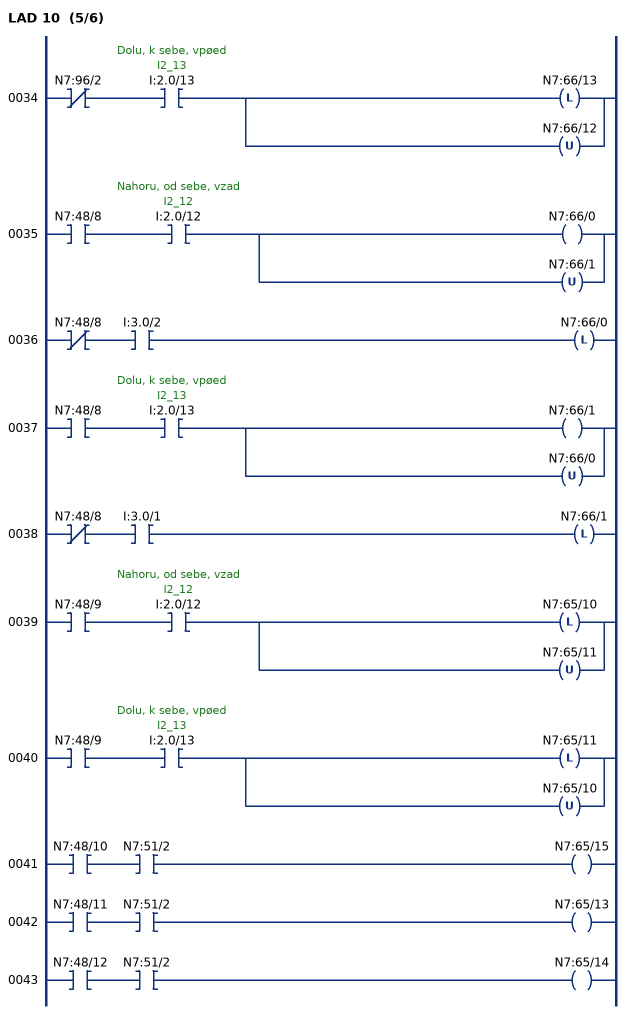
% Rung: 34 %
SOR XIO N7:96/2 XIC I:2.0/13 BST OTL N7:66/13 NXB OTU N7:66/12 BND EOR
%   I:2.0/13  I2_13  "Dolu, k sebe, vpøed" %
% Rung: 35 %
SOR XIC N7:48/8 XIC I:2.0/12 BST OTE N7:66/0 NXB OTU N7:66/1 BND EOR
%   I:2.0/12  I2_12  "Nahoru, od sebe, vzad" %
% Rung: 36 %
SOR XIO N7:48/8 XIC I:3.0/2 OTL N7:66/0 EOR
% Rung: 37 %
SOR XIC N7:48/8 XIC I:2.0/13 BST OTE N7:66/1 NXB OTU N7:66/0 BND EOR
%   I:2.0/13  I2_13  "Dolu, k sebe, vpøed" %
% Rung: 38 %
SOR XIO N7:48/8 XIC I:3.0/1 OTL N7:66/1 EOR
% Rung: 39 %
SOR XIC N7:48/9 XIC I:2.0/12 BST OTL N7:65/10 NXB OTU N7:65/11 BND EOR
%   I:2.0/12  I2_12  "Nahoru, od sebe, vzad" %
% Rung: 40 %
SOR XIC N7:48/9 XIC I:2.0/13 BST OTL N7:65/11 NXB OTU N7:65/10 BND EOR
%   I:2.0/13  I2_13  "Dolu, k sebe, vpøed" %
% Rung: 41 %
SOR XIC N7:48/10 XIC N7:51/2 OTE N7:65/15 EOR
% Rung: 42 %
SOR XIC N7:48/11 XIC N7:51/2 OTE N7:65/13 EOR
% Rung: 43 %
SOR XIC N7:48/12 XIC N7:51/2 OTE N7:65/14 EOR

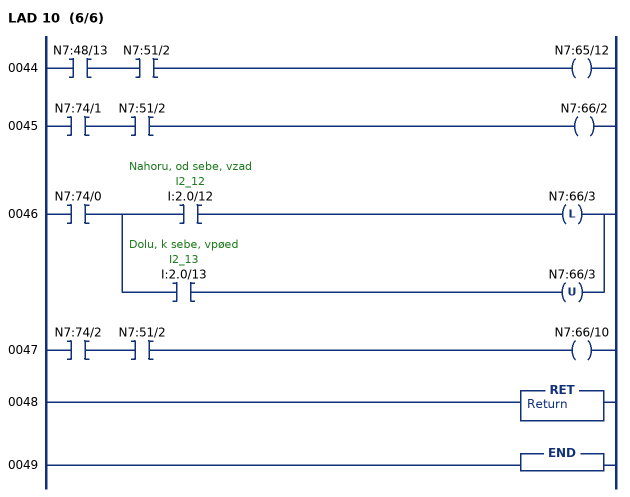
% Rung: 44 %
SOR XIC N7:48/13 XIC N7:51/2 OTE N7:65/12 EOR
% Rung: 45 %
SOR XIC N7:74/1 XIC N7:51/2 OTE N7:66/2 EOR
% Rung: 46 %
SOR XIC N7:74/0 BST XIC I:2.0/12 OTL N7:66/3 NXB XIC I:2.0/13 OTU N7:66/3 BND EOR
%   I:2.0/12  I2_12  "Nahoru, od sebe, vzad" %
%   I:2.0/13  I2_13  "Dolu, k sebe, vpøed" %
% Rung: 47 %
SOR XIC N7:74/2 XIC N7:51/2 OTE N7:66/10 EOR
% Rung: 48 %
SOR RET EOR
% Rung: 49 %
SOR END EOR

LADDER 11
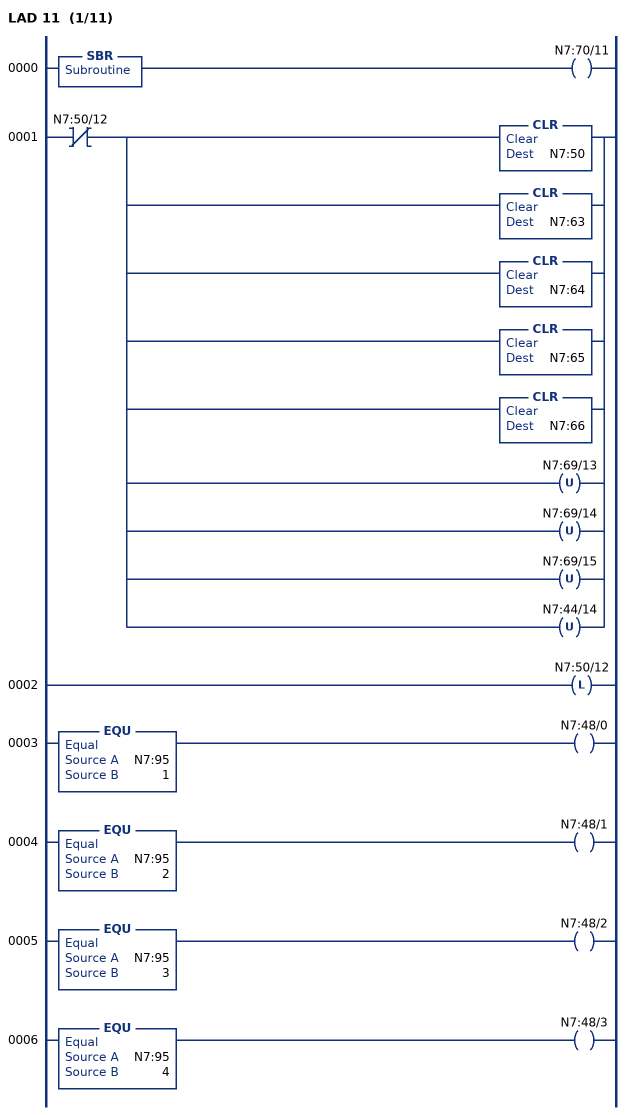
% Rung: 0 %
SOR SBR OTE N7:70/11 EOR
% Rung: 1 %
SOR XIO N7:50/12 BST CLR N7:50 NXB CLR N7:63 NXB CLR N7:64 NXB CLR N7:65 NXB CLR N7:66 NXB OTU N7:69/13 NXB OTU N7:69/14 NXB OTU N7:69/15 NXB OTU N7:44/14 BND EOR
% Rung: 2 %
SOR OTL N7:50/12 EOR
% Rung: 3 %
SOR EQU N7:95 1 OTE N7:48/0 EOR
% Rung: 4 %
SOR EQU N7:95 2 OTE N7:48/1 EOR
% Rung: 5 %
SOR EQU N7:95 3 OTE N7:48/2 EOR
% Rung: 6 %
SOR EQU N7:95 4 OTE N7:48/3 EOR

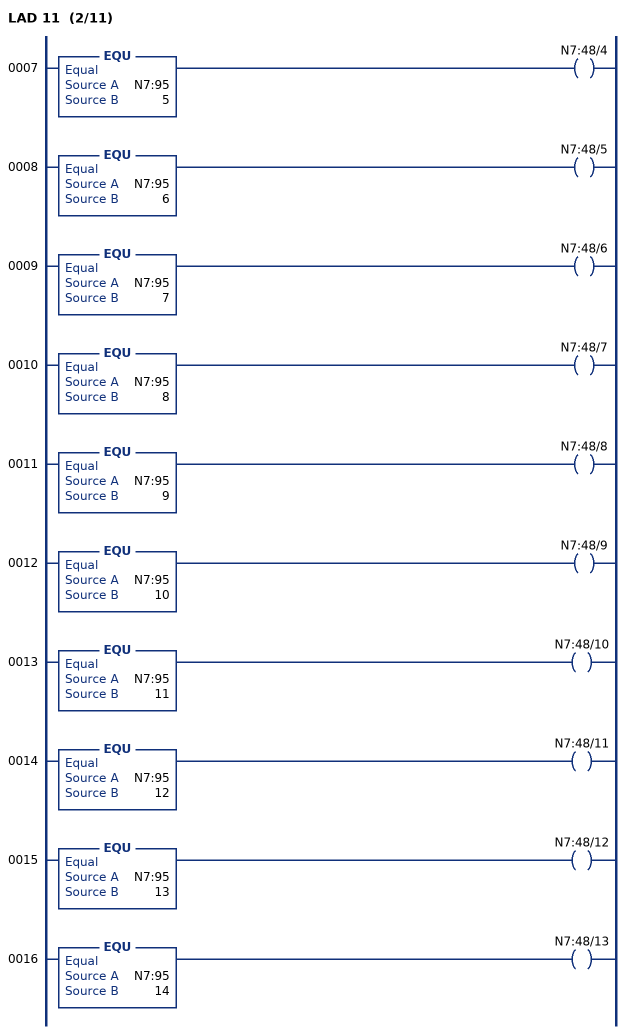
% Rung: 7 %
SOR EQU N7:95 5 OTE N7:48/4 EOR
% Rung: 8 %
SOR EQU N7:95 6 OTE N7:48/5 EOR
% Rung: 9 %
SOR EQU N7:95 7 OTE N7:48/6 EOR
% Rung: 10 %
SOR EQU N7:95 8 OTE N7:48/7 EOR
% Rung: 11 %
SOR EQU N7:95 9 OTE N7:48/8 EOR
% Rung: 12 %
SOR EQU N7:95 10 OTE N7:48/9 EOR
% Rung: 13 %
SOR EQU N7:95 11 OTE N7:48/10 EOR
% Rung: 14 %
SOR EQU N7:95 12 OTE N7:48/11 EOR
% Rung: 15 %
SOR EQU N7:95 13 OTE N7:48/12 EOR
% Rung: 16 %
SOR EQU N7:95 14 OTE N7:48/13 EOR

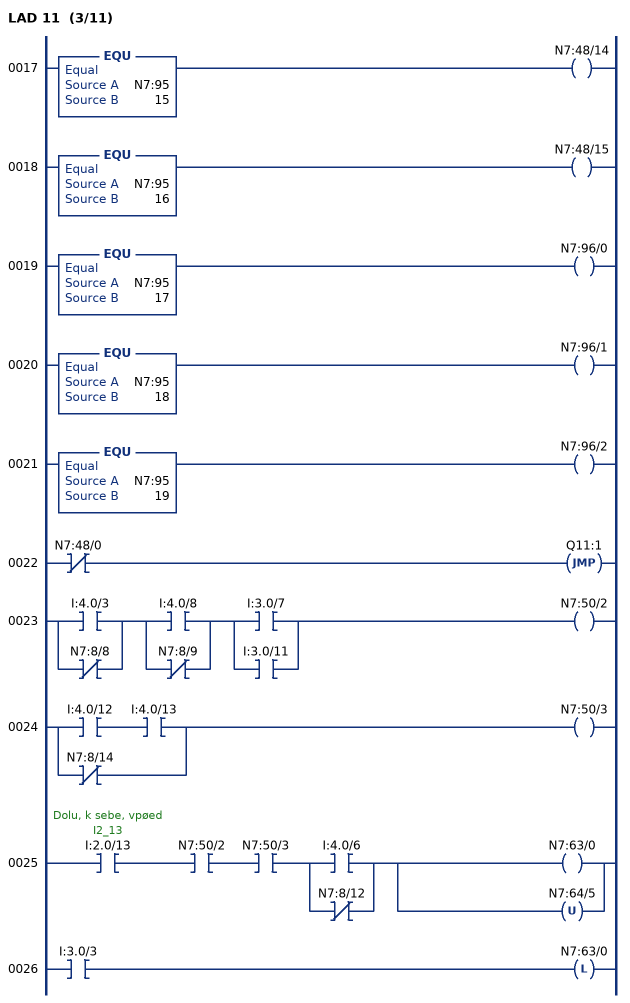
% Rung: 17 %
SOR EQU N7:95 15 OTE N7:48/14 EOR
% Rung: 18 %
SOR EQU N7:95 16 OTE N7:48/15 EOR
% Rung: 19 %
SOR EQU N7:95 17 OTE N7:96/0 EOR
% Rung: 20 %
SOR EQU N7:95 18 OTE N7:96/1 EOR
% Rung: 21 %
SOR EQU N7:95 19 OTE N7:96/2 EOR
% Rung: 22 %
SOR XIO N7:48/0 JMP Q11:1 EOR
% Rung: 23 %
SOR BST XIC I:4.0/3 NXB XIO N7:8/8 BND BST XIC I:4.0/8 NXB XIO N7:8/9 BND BST XIC I:3.0/7 NXB XIC I:3.0/11 BND OTE N7:50/2 EOR
% Rung: 24 %
SOR BST XIC I:4.0/12 XIC I:4.0/13 NXB XIO N7:8/14 BND OTE N7:50/3 EOR
% Rung: 25 %
SOR XIC I:2.0/13 XIC N7:50/2 XIC N7:50/3 BST XIC I:4.0/6 NXB XIO N7:8/12 BND BST OTE N7:63/0 NXB OTU N7:64/5 BND EOR
%   I:2.0/13  I2_13  "Dolu, k sebe, vpøed" %
% Rung: 26 %
SOR XIC I:3.0/3 OTL N7:63/0 EOR

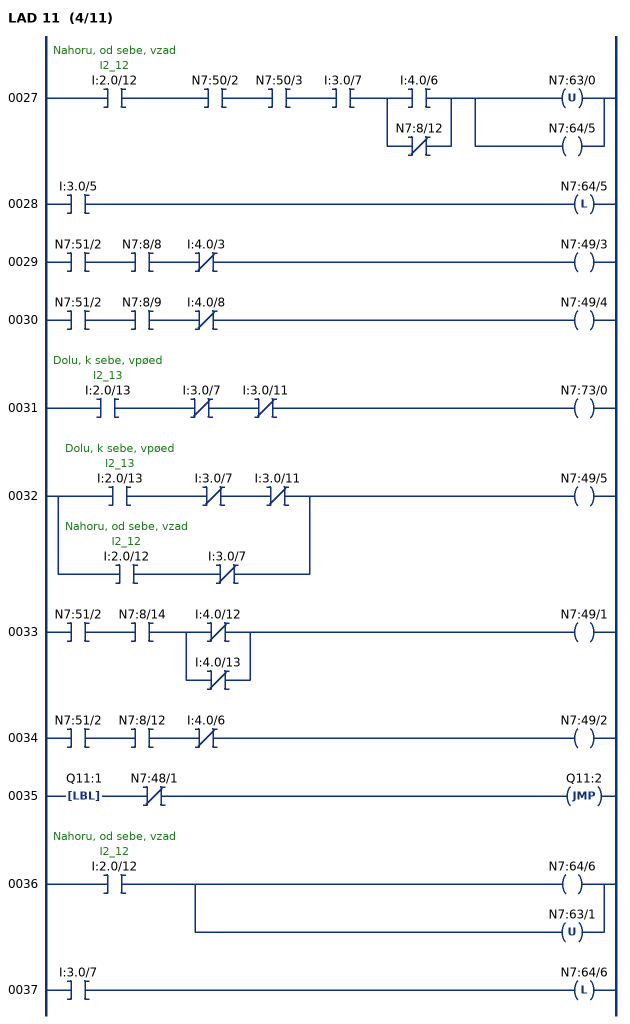
% Rung: 27 %
SOR XIC I:2.0/12 XIC N7:50/2 XIC N7:50/3 XIC I:3.0/7 BST XIC I:4.0/6 NXB XIO N7:8/12 BND BST OTU N7:63/0 NXB OTE N7:64/5 BND EOR
%   I:2.0/12  I2_12  "Nahoru, od sebe, vzad" %
% Rung: 28 %
SOR XIC I:3.0/5 OTL N7:64/5 EOR
% Rung: 29 %
SOR XIC N7:51/2 XIC N7:8/8 XIO I:4.0/3 OTE N7:49/3 EOR
% Rung: 30 %
SOR XIC N7:51/2 XIC N7:8/9 XIO I:4.0/8 OTE N7:49/4 EOR
% Rung: 31 %
SOR XIC I:2.0/13 XIO I:3.0/7 XIO I:3.0/11 OTE N7:73/0 EOR
%   I:2.0/13  I2_13  "Dolu, k sebe, vpøed" %
% Rung: 32 %
SOR BST XIC I:2.0/13 XIO I:3.0/7 XIO I:3.0/11 NXB XIC I:2.0/12 XIO I:3.0/7 BND OTE N7:49/5 EOR
%   I:2.0/13  I2_13  "Dolu, k sebe, vpøed" %
%   I:2.0/12  I2_12  "Nahoru, od sebe, vzad" %
% Rung: 33 %
SOR XIC N7:51/2 XIC N7:8/14 BST XIO I:4.0/12 NXB XIO I:4.0/13 BND OTE N7:49/1 EOR
% Rung: 34 %
SOR XIC N7:51/2 XIC N7:8/12 XIO I:4.0/6 OTE N7:49/2 EOR
% Rung: 35 %
SOR LBL Q11:1 XIO N7:48/1 JMP Q11:2 EOR
% Rung: 36 %
SOR XIC I:2.0/12 BST OTE N7:64/6 NXB OTU N7:63/1 BND EOR
%   I:2.0/12  I2_12  "Nahoru, od sebe, vzad" %
% Rung: 37 %
SOR XIC I:3.0/7 OTL N7:64/6 EOR

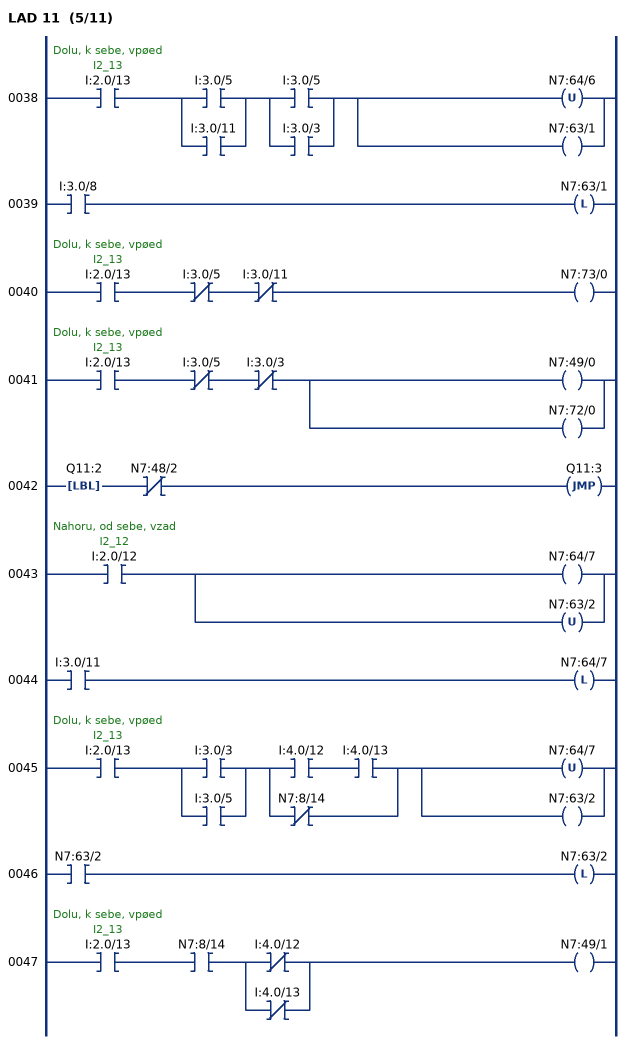
% Rung: 38 %
SOR XIC I:2.0/13 BST XIC I:3.0/5 NXB XIC I:3.0/11 BND BST XIC I:3.0/5 NXB XIC I:3.0/3 BND BST OTU N7:64/6 NXB OTE N7:63/1 BND EOR
%   I:2.0/13  I2_13  "Dolu, k sebe, vpøed" %
% Rung: 39 %
SOR XIC I:3.0/8 OTL N7:63/1 EOR
% Rung: 40 %
SOR XIC I:2.0/13 XIO I:3.0/5 XIO I:3.0/11 OTE N7:73/0 EOR
%   I:2.0/13  I2_13  "Dolu, k sebe, vpøed" %
% Rung: 41 %
SOR XIC I:2.0/13 XIO I:3.0/5 XIO I:3.0/3 BST OTE N7:49/0 NXB OTE N7:72/0 BND EOR
%   I:2.0/13  I2_13  "Dolu, k sebe, vpøed" %
% Rung: 42 %
SOR LBL Q11:2 XIO N7:48/2 JMP Q11:3 EOR
% Rung: 43 %
SOR XIC I:2.0/12 BST OTE N7:64/7 NXB OTU N7:63/2 BND EOR
%   I:2.0/12  I2_12  "Nahoru, od sebe, vzad" %
% Rung: 44 %
SOR XIC I:3.0/11 OTL N7:64/7 EOR
% Rung: 45 %
SOR XIC I:2.0/13 BST XIC I:3.0/3 NXB XIC I:3.0/5 BND BST XIC I:4.0/12 XIC I:4.0/13 NXB XIO N7:8/14 BND BST OTU N7:64/7 NXB OTE N7:63/2 BND EOR
%   I:2.0/13  I2_13  "Dolu, k sebe, vpøed" %
% Rung: 46 %
SOR XIC N7:63/2 OTL N7:63/2 EOR
% Rung: 47 %
SOR XIC I:2.0/13 XIC N7:8/14 BST XIO I:4.0/12 NXB XIO I:4.0/13 BND OTE N7:49/1 EOR
%   I:2.0/13  I2_13  "Dolu, k sebe, vpøed" %

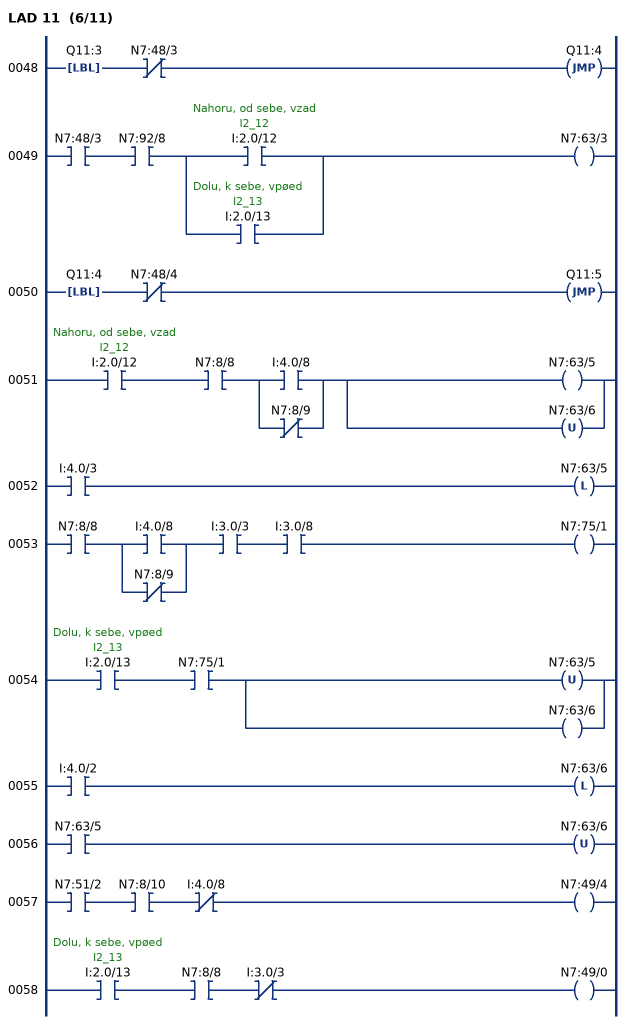
% Rung: 48 %
SOR LBL Q11:3 XIO N7:48/3 JMP Q11:4 EOR
% Rung: 49 %
SOR XIC N7:48/3 XIC N7:92/8 BST XIC I:2.0/12 NXB XIC I:2.0/13 BND OTE N7:63/3 EOR
%   I:2.0/12  I2_12  "Nahoru, od sebe, vzad" %
%   I:2.0/13  I2_13  "Dolu, k sebe, vpøed" %
% Rung: 50 %
SOR LBL Q11:4 XIO N7:48/4 JMP Q11:5 EOR
% Rung: 51 %
SOR XIC I:2.0/12 XIC N7:8/8 BST XIC I:4.0/8 NXB XIO N7:8/9 BND BST OTE N7:63/5 NXB OTU N7:63/6 BND EOR
%   I:2.0/12  I2_12  "Nahoru, od sebe, vzad" %
% Rung: 52 %
SOR XIC I:4.0/3 OTL N7:63/5 EOR
% Rung: 53 %
SOR XIC N7:8/8 BST XIC I:4.0/8 NXB XIO N7:8/9 BND XIC I:3.0/3 XIC I:3.0/8 OTE N7:75/1 EOR
% Rung: 54 %
SOR XIC I:2.0/13 XIC N7:75/1 BST OTU N7:63/5 NXB OTE N7:63/6 BND EOR
%   I:2.0/13  I2_13  "Dolu, k sebe, vpøed" %
% Rung: 55 %
SOR XIC I:4.0/2 OTL N7:63/6 EOR
% Rung: 56 %
SOR XIC N7:63/5 OTU N7:63/6 EOR
% Rung: 57 %
SOR XIC N7:51/2 XIC N7:8/10 XIO I:4.0/8 OTE N7:49/4 EOR
% Rung: 58 %
SOR XIC I:2.0/13 XIC N7:8/8 XIO I:3.0/3 OTE N7:49/0 EOR
%   I:2.0/13  I2_13  "Dolu, k sebe, vpøed" %

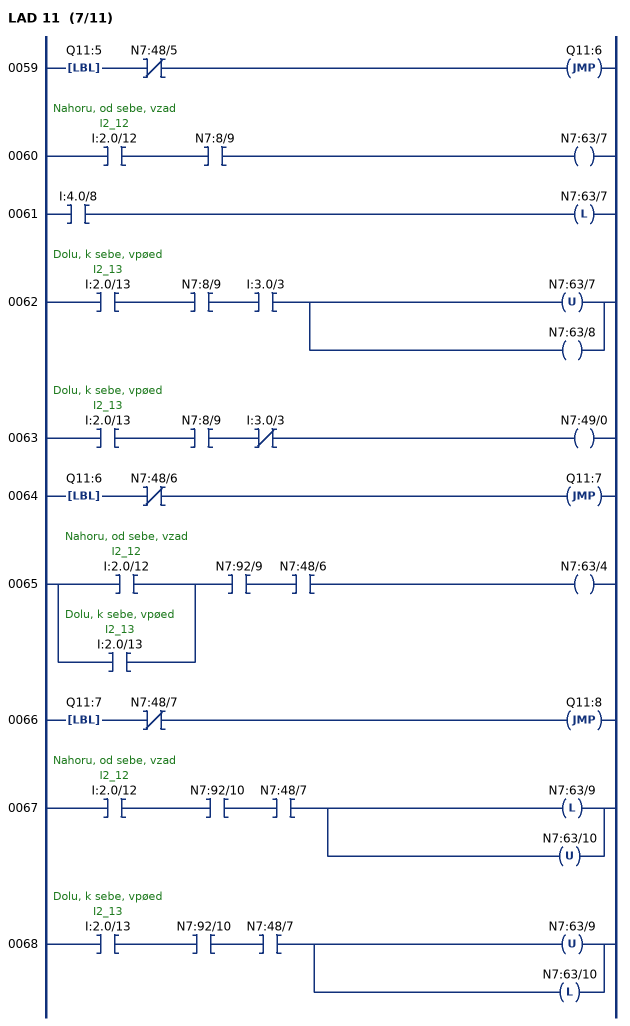
% Rung: 59 %
SOR LBL Q11:5 XIO N7:48/5 JMP Q11:6 EOR
% Rung: 60 %
SOR XIC I:2.0/12 XIC N7:8/9 OTE N7:63/7 EOR
%   I:2.0/12  I2_12  "Nahoru, od sebe, vzad" %
% Rung: 61 %
SOR XIC I:4.0/8 OTL N7:63/7 EOR
% Rung: 62 %
SOR XIC I:2.0/13 XIC N7:8/9 XIC I:3.0/3 BST OTU N7:63/7 NXB OTE N7:63/8 BND EOR
%   I:2.0/13  I2_13  "Dolu, k sebe, vpøed" %
% Rung: 63 %
SOR XIC I:2.0/13 XIC N7:8/9 XIO I:3.0/3 OTE N7:49/0 EOR
%   I:2.0/13  I2_13  "Dolu, k sebe, vpøed" %
% Rung: 64 %
SOR LBL Q11:6 XIO N7:48/6 JMP Q11:7 EOR
% Rung: 65 %
SOR BST XIC I:2.0/12 NXB XIC I:2.0/13 BND XIC N7:92/9 XIC N7:48/6 OTE N7:63/4 EOR
%   I:2.0/12  I2_12  "Nahoru, od sebe, vzad" %
%   I:2.0/13  I2_13  "Dolu, k sebe, vpøed" %
% Rung: 66 %
SOR LBL Q11:7 XIO N7:48/7 JMP Q11:8 EOR
% Rung: 67 %
SOR XIC I:2.0/12 XIC N7:92/10 XIC N7:48/7 BST OTL N7:63/9 NXB OTU N7:63/10 BND EOR
%   I:2.0/12  I2_12  "Nahoru, od sebe, vzad" %
% Rung: 68 %
SOR XIC I:2.0/13 XIC N7:92/10 XIC N7:48/7 BST OTU N7:63/9 NXB OTL N7:63/10 BND EOR
%   I:2.0/13  I2_13  "Dolu, k sebe, vpøed" %

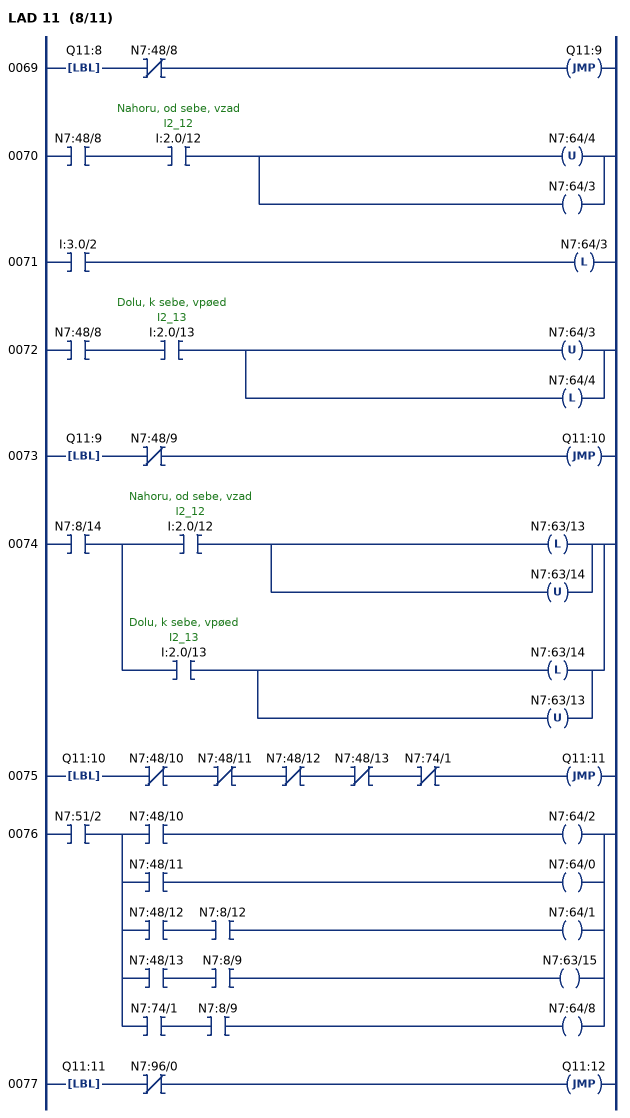
% Rung: 69 %
SOR LBL Q11:8 XIO N7:48/8 JMP Q11:9 EOR
% Rung: 70 %
SOR XIC N7:48/8 XIC I:2.0/12 BST OTU N7:64/4 NXB OTE N7:64/3 BND EOR
%   I:2.0/12  I2_12  "Nahoru, od sebe, vzad" %
% Rung: 71 %
SOR XIC I:3.0/2 OTL N7:64/3 EOR
% Rung: 72 %
SOR XIC N7:48/8 XIC I:2.0/13 BST OTU N7:64/3 NXB OTL N7:64/4 BND EOR
%   I:2.0/13  I2_13  "Dolu, k sebe, vpøed" %
% Rung: 73 %
SOR LBL Q11:9 XIO N7:48/9 JMP Q11:10 EOR
% Rung: 74 %
SOR XIC N7:8/14 BST XIC I:2.0/12 BST OTL N7:63/13 NXB OTU N7:63/14 BND NXB XIC I:2.0/13 BST OTL N7:63/14 NXB OTU N7:63/13 BND BND EOR
%   I:2.0/12  I2_12  "Nahoru, od sebe, vzad" %
%   I:2.0/13  I2_13  "Dolu, k sebe, vpøed" %
% Rung: 75 %
SOR LBL Q11:10 XIO N7:48/10 XIO N7:48/11 XIO N7:48/12 XIO N7:48/13 XIO N7:74/1 JMP Q11:11 EOR
% Rung: 76 %
SOR XIC N7:51/2 BST XIC N7:48/10 OTE N7:64/2 NXB BST XIC N7:48/11 OTE N7:64/0 NXB XIC N7:48/12 XIC N7:8/12 OTE N7:64/1 NXB XIC N7:48/13 XIC N7:8/9 OTE N7:63/15 NXB XIC N7:74/1 XIC N7:8/9 OTE N7:64/8 BND BND EOR
% Rung: 77 %
SOR LBL Q11:11 XIO N7:96/0 JMP Q11:12 EOR

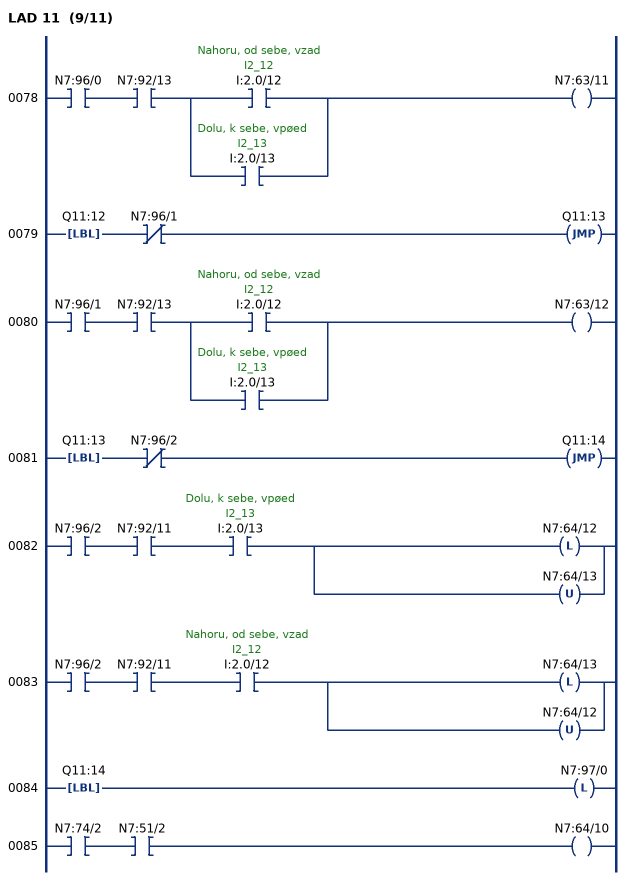
% Rung: 78 %
SOR XIC N7:96/0 XIC N7:92/13 BST XIC I:2.0/12 NXB XIC I:2.0/13 BND OTE N7:63/11 EOR
%   I:2.0/12  I2_12  "Nahoru, od sebe, vzad" %
%   I:2.0/13  I2_13  "Dolu, k sebe, vpøed" %
% Rung: 79 %
SOR LBL Q11:12 XIO N7:96/1 JMP Q11:13 EOR
% Rung: 80 %
SOR XIC N7:96/1 XIC N7:92/13 BST XIC I:2.0/12 NXB XIC I:2.0/13 BND OTE N7:63/12 EOR
%   I:2.0/12  I2_12  "Nahoru, od sebe, vzad" %
%   I:2.0/13  I2_13  "Dolu, k sebe, vpøed" %
% Rung: 81 %
SOR LBL Q11:13 XIO N7:96/2 JMP Q11:14 EOR
% Rung: 82 %
SOR XIC N7:96/2 XIC N7:92/11 XIC I:2.0/13 BST OTL N7:64/12 NXB OTU N7:64/13 BND EOR
%   I:2.0/13  I2_13  "Dolu, k sebe, vpøed" %
% Rung: 83 %
SOR XIC N7:96/2 XIC N7:92/11 XIC I:2.0/12 BST OTL N7:64/13 NXB OTU N7:64/12 BND EOR
%   I:2.0/12  I2_12  "Nahoru, od sebe, vzad" %
% Rung: 84 %
SOR LBL Q11:14 OTL N7:97/0 EOR
% Rung: 85 %
SOR XIC N7:74/2 XIC N7:51/2 OTE N7:64/10 EOR

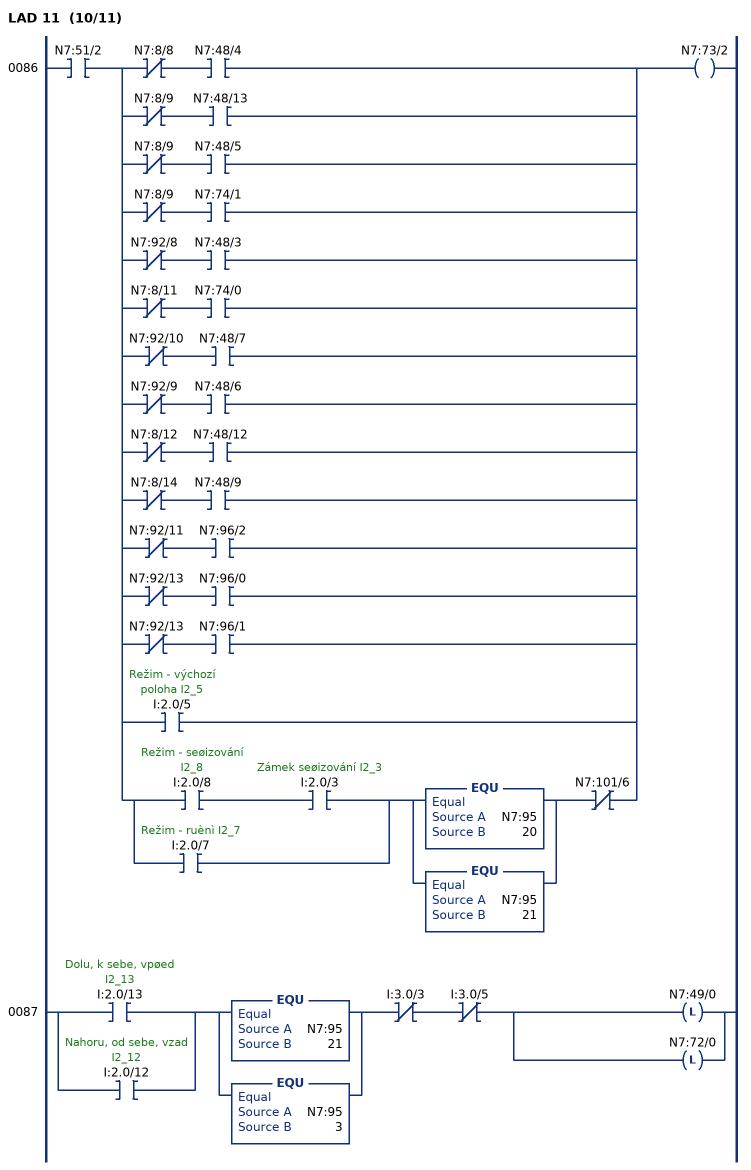
% Rung: 86 %
SOR XIC N7:51/2 BST XIO N7:8/8 XIC N7:48/4 NXB XIO N7:8/9 XIC N7:48/13 NXB XIO N7:8/9 XIC N7:48/5 NXB XIO N7:8/9 XIC N7:74/1 NXB XIO N7:92/8 XIC N7:48/3 NXB XIO N7:8/11 XIC N7:74/0 NXB XIO N7:92/10 XIC N7:48/7 NXB XIO N7:92/9 XIC N7:48/6 NXB XIO N7:8/12 XIC N7:48/12 NXB BST BST BST XIO N7:8/14 XIC N7:48/9 NXB XIO N7:92/11 XIC N7:96/2 BND NXB XIO N7:92/13 XIC N7:96/0 BND NXB XIO N7:92/13 XIC N7:96/1 NXB BST XIC I:2.0/5 NXB BST XIC I:2.0/8 XIC I:2.0/3 NXB XIC I:2.0/7 BND BST EQU N7:95 20 NXB EQU N7:95 21 BND XIO N7:101/6 BND BND BND OTE N7:73/2 EOR
%   I:2.0/5  I2_5  "Režim - výchozí poloha" %
%   I:2.0/8  I2_8  "Režim - seøizování" %
%   I:2.0/3  I2_3  "Zámek seøizování" %
%   I:2.0/7  I2_7  "Režim - ruènì" %
% Rung: 87 %
SOR BST XIC I:2.0/13 NXB XIC I:2.0/12 BND BST EQU N7:95 21 NXB EQU N7:95 3 BND XIO I:3.0/3 XIO I:3.0/5 BST OTL N7:49/0 NXB OTL N7:72/0 BND EOR
%   I:2.0/13  I2_13  "Dolu, k sebe, vpøed" %
%   I:2.0/12  I2_12  "Nahoru, od sebe, vzad" %

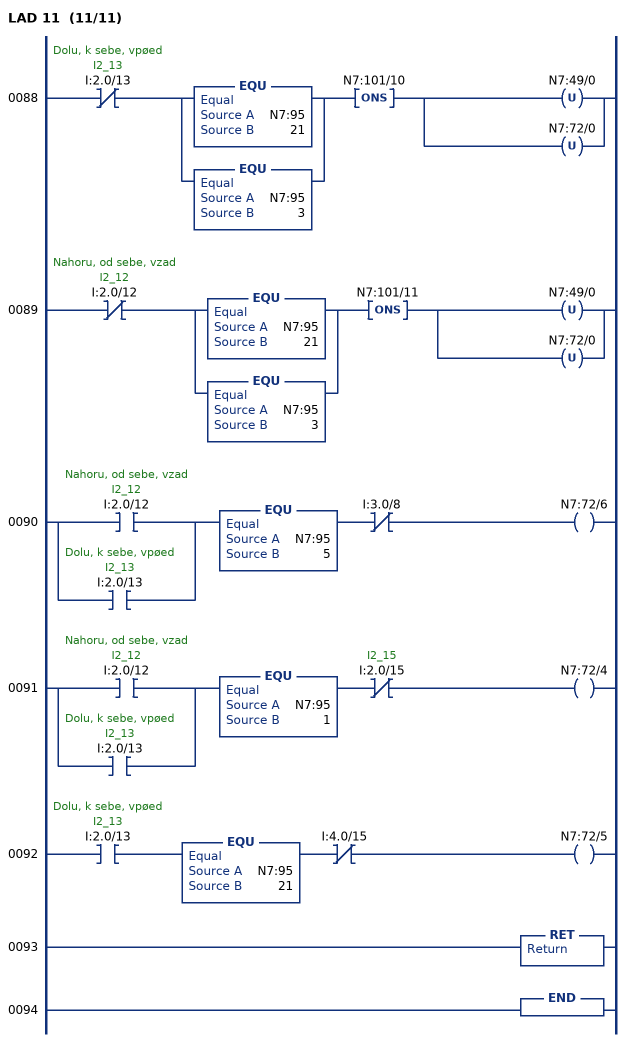
% Rung: 88 %
SOR XIO I:2.0/13 BST EQU N7:95 21 NXB EQU N7:95 3 BND OSR N7:101/10 BST OTU N7:49/0 NXB OTU N7:72/0 BND EOR
%   I:2.0/13  I2_13  "Dolu, k sebe, vpøed" %
% Rung: 89 %
SOR XIO I:2.0/12 BST EQU N7:95 21 NXB EQU N7:95 3 BND OSR N7:101/11 BST OTU N7:49/0 NXB OTU N7:72/0 BND EOR
%   I:2.0/12  I2_12  "Nahoru, od sebe, vzad" %
% Rung: 90 %
SOR BST XIC I:2.0/12 NXB XIC I:2.0/13 BND EQU N7:95 5 XIO I:3.0/8 OTE N7:72/6 EOR
%   I:2.0/12  I2_12  "Nahoru, od sebe, vzad" %
%   I:2.0/13  I2_13  "Dolu, k sebe, vpøed" %
% Rung: 91 %
SOR BST XIC I:2.0/12 NXB XIC I:2.0/13 BND EQU N7:95 1 XIO I:2.0/15 OTE N7:72/4 EOR
%   I:2.0/12  I2_12  "Nahoru, od sebe, vzad" %
%   I:2.0/13  I2_13  "Dolu, k sebe, vpøed" %
%   I:2.0/15  I2_15 %
% Rung: 92 %
SOR XIC I:2.0/13 EQU N7:95 21 XIO I:4.0/15 OTE N7:72/5 EOR
%   I:2.0/13  I2_13  "Dolu, k sebe, vpøed" %
% Rung: 93 %
SOR RET EOR
% Rung: 94 %
SOR END EOR

LADDER 12
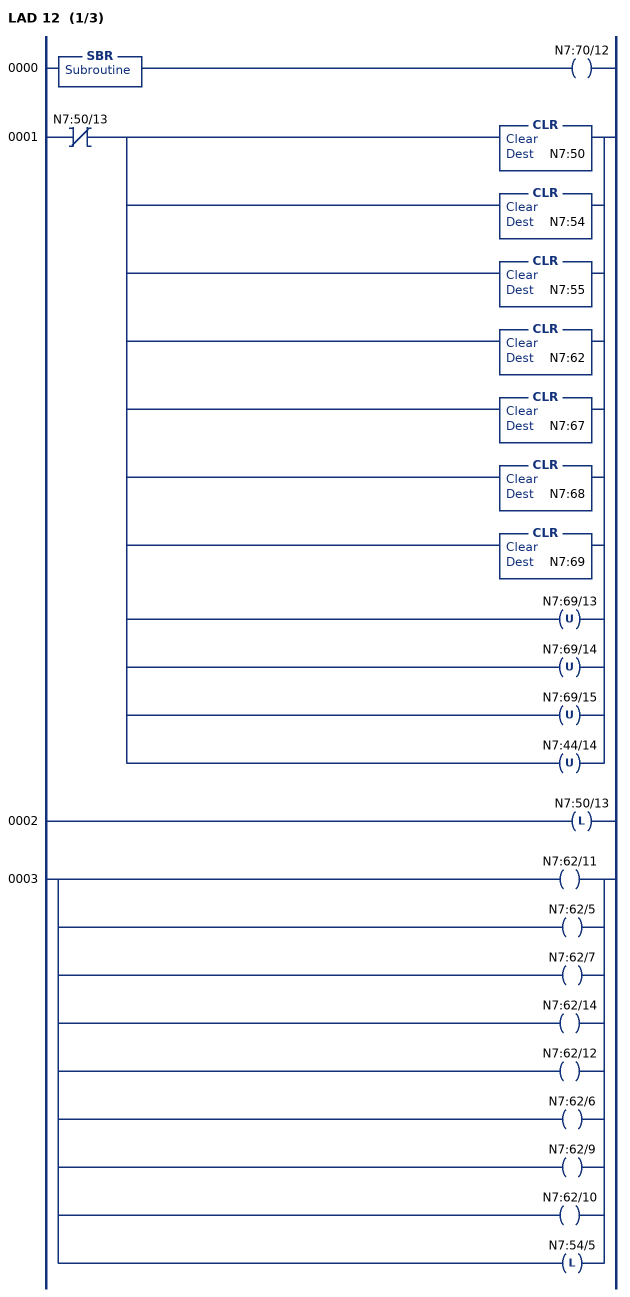
% Rung: 0 %
SOR SBR OTE N7:70/12 EOR
% Rung: 1 %
SOR XIO N7:50/13 BST CLR N7:50 NXB CLR N7:54 NXB CLR N7:55 NXB CLR N7:62 NXB CLR N7:67 NXB CLR N7:68 NXB CLR N7:69 NXB OTU N7:69/13 NXB OTU N7:69/14 NXB OTU N7:69/15 NXB OTU N7:44/14 BND EOR
% Rung: 2 %
SOR OTL N7:50/13 EOR
% Rung: 3 %
SOR BST OTE N7:62/11 NXB OTE N7:62/5 NXB OTE N7:62/7 NXB OTE N7:62/14 NXB BST OTE N7:62/12 NXB OTE N7:62/6 BND NXB OTE N7:62/9 NXB OTE N7:62/10 NXB OTL N7:54/5 BND EOR

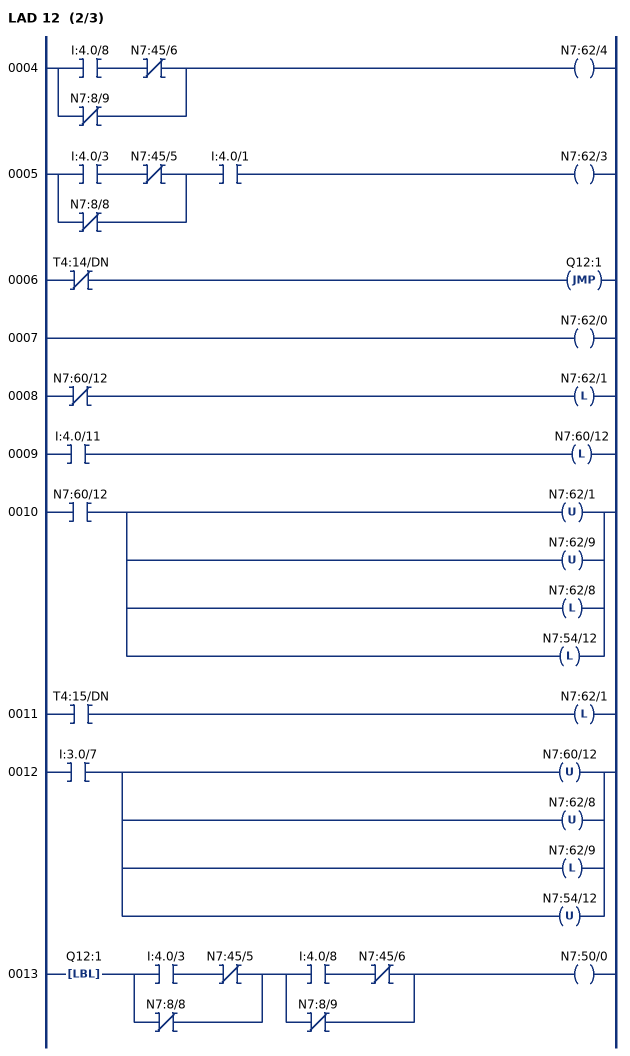
% Rung: 4 %
SOR BST XIC I:4.0/8 XIO N7:45/6 NXB XIO N7:8/9 BND OTE N7:62/4 EOR
% Rung: 5 %
SOR BST XIC I:4.0/3 XIO N7:45/5 NXB XIO N7:8/8 BND XIC I:4.0/1 OTE N7:62/3 EOR
% Rung: 6 %
SOR XIO T4:14/DN JMP Q12:1 EOR
% Rung: 7 %
SOR OTE N7:62/0 EOR
% Rung: 8 %
SOR XIO N7:60/12 OTL N7:62/1 EOR
% Rung: 9 %
SOR XIC I:4.0/11 OTL N7:60/12 EOR
% Rung: 10 %
SOR XIC N7:60/12 BST OTU N7:62/1 NXB BST OTU N7:62/9 NXB OTL N7:62/8 NXB OTL N7:54/12 BND BND EOR
% Rung: 11 %
SOR XIC T4:15/DN OTL N7:62/1 EOR
% Rung: 12 %
SOR XIC I:3.0/7 BST OTU N7:60/12 NXB OTU N7:62/8 NXB OTL N7:62/9 NXB OTU N7:54/12 BND EOR
% Rung: 13 %
SOR LBL Q12:1 BST XIC I:4.0/3 XIO N7:45/5 NXB XIO N7:8/8 BND BST XIC I:4.0/8 XIO N7:45/6 NXB XIO N7:8/9 BND OTE N7:50/0 EOR

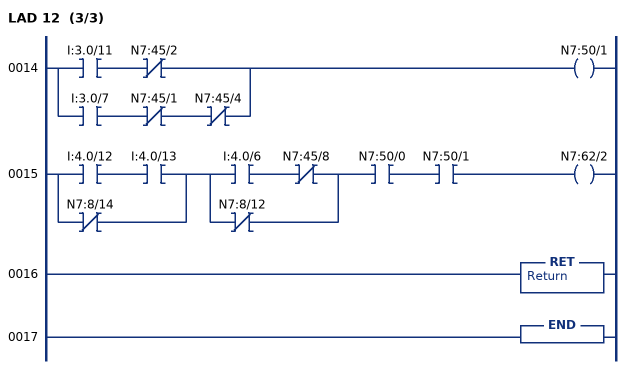
% Rung: 14 %
SOR BST XIC I:3.0/11 XIO N7:45/2 NXB XIC I:3.0/7 XIO N7:45/1 XIO N7:45/4 BND OTE N7:50/1 EOR
% Rung: 15 %
SOR BST XIC I:4.0/12 XIC I:4.0/13 NXB XIO N7:8/14 BND BST XIC I:4.0/6 XIO N7:45/8 NXB XIO N7:8/12 BND XIC N7:50/0 XIC N7:50/1 OTE N7:62/2 EOR
% Rung: 16 %
SOR RET EOR
% Rung: 17 %
SOR END EOR

LADDER 13
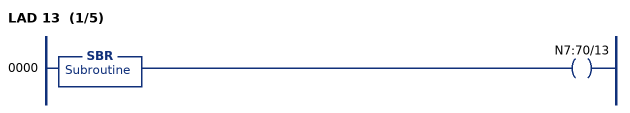
% Rung: 0 %
SOR SBR OTE N7:70/13 EOR

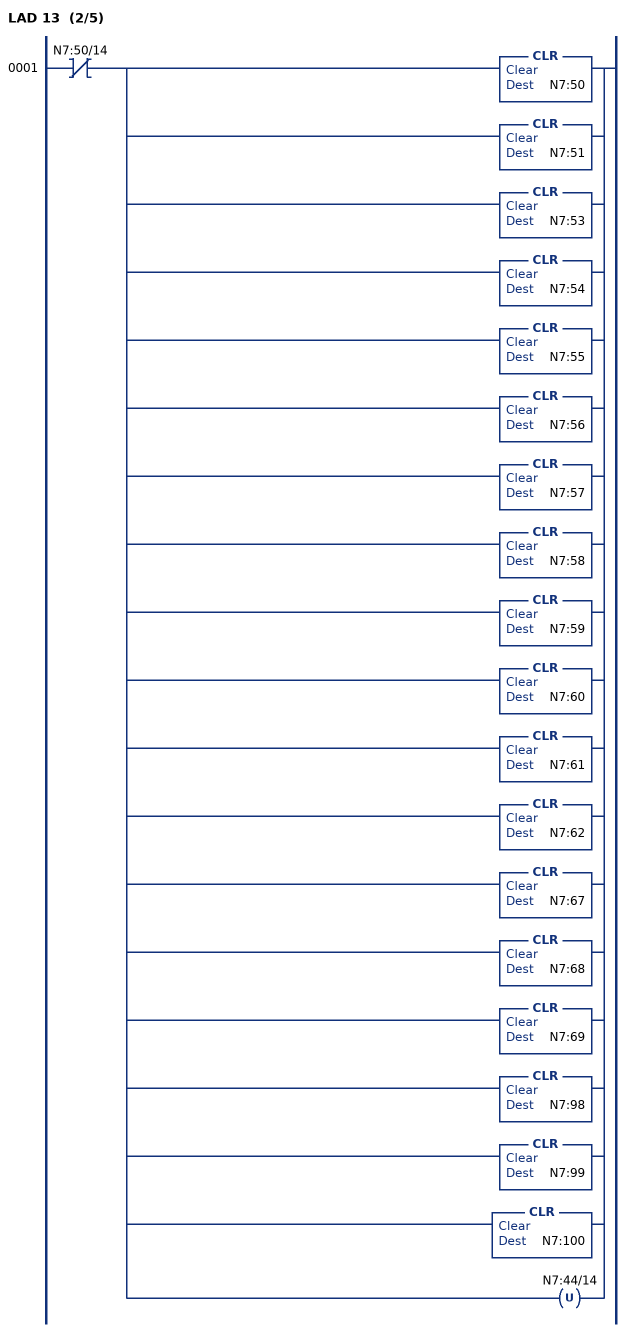
% Rung: 1 %
SOR XIO N7:50/14 BST CLR N7:50 NXB CLR N7:51 NXB CLR N7:53 NXB CLR N7:54 NXB CLR N7:55 NXB CLR N7:56 NXB CLR N7:57 NXB CLR N7:58 NXB CLR N7:59 NXB CLR N7:60 NXB CLR N7:61 NXB CLR N7:62 NXB CLR N7:67 NXB CLR N7:68 NXB BST BST CLR N7:69 NXB CLR N7:98 BND NXB BST CLR N7:99 NXB CLR N7:100 BND BND NXB OTU N7:44/14 BND EOR

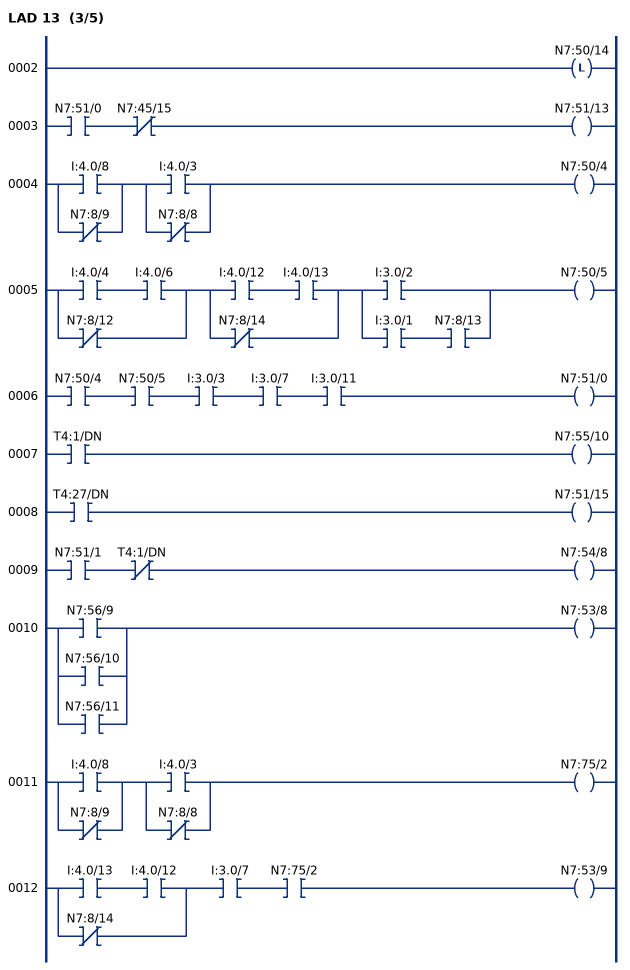
% Rung: 2 %
SOR OTL N7:50/14 EOR
% Rung: 3 %
SOR XIC N7:51/0 XIO N7:45/15 OTE N7:51/13 EOR
% Rung: 4 %
SOR BST XIC I:4.0/8 NXB XIO N7:8/9 BND BST XIC I:4.0/3 NXB XIO N7:8/8 BND OTE N7:50/4 EOR
% Rung: 5 %
SOR BST XIC I:4.0/4 XIC I:4.0/6 NXB XIO N7:8/12 BND BST XIC I:4.0/12 XIC I:4.0/13 NXB XIO N7:8/14 BND BST XIC I:3.0/2 NXB XIC I:3.0/1 XIC N7:8/13 BND OTE N7:50/5 EOR
% Rung: 6 %
SOR XIC N7:50/4 XIC N7:50/5 XIC I:3.0/3 XIC I:3.0/7 XIC I:3.0/11 OTE N7:51/0 EOR
% Rung: 7 %
SOR XIC T4:1/DN OTE N7:55/10 EOR
% Rung: 8 %
SOR XIC T4:27/DN OTE N7:51/15 EOR
% Rung: 9 %
SOR XIC N7:51/1 XIO T4:1/DN OTE N7:54/8 EOR
% Rung: 10 %
SOR BST XIC N7:56/9 NXB XIC N7:56/10 NXB XIC N7:56/11 BND OTE N7:53/8 EOR
% Rung: 11 %
SOR BST XIC I:4.0/8 NXB XIO N7:8/9 BND BST XIC I:4.0/3 NXB XIO N7:8/8 BND OTE N7:75/2 EOR
% Rung: 12 %
SOR BST XIC I:4.0/13 XIC I:4.0/12 NXB XIO N7:8/14 BND XIC I:3.0/7 XIC N7:75/2 OTE N7:53/9 EOR

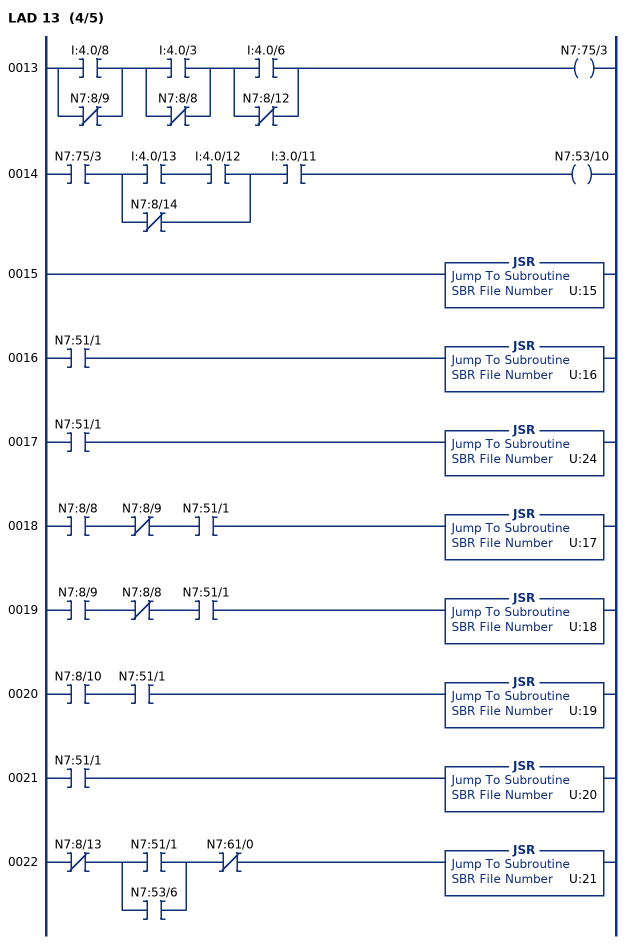
% Rung: 13 %
SOR BST XIC I:4.0/8 NXB XIO N7:8/9 BND BST XIC I:4.0/3 NXB XIO N7:8/8 BND BST XIC I:4.0/6 NXB XIO N7:8/12 BND OTE N7:75/3 EOR
% Rung: 14 %
SOR XIC N7:75/3 BST XIC I:4.0/13 XIC I:4.0/12 NXB XIO N7:8/14 BND XIC I:3.0/11 OTE N7:53/10 EOR
% Rung: 15 %
SOR JSR U:15 EOR
% Rung: 16 %
SOR XIC N7:51/1 JSR U:16 EOR
% Rung: 17 %
SOR XIC N7:51/1 JSR U:24 EOR
% Rung: 18 %
SOR XIC N7:8/8 XIO N7:8/9 XIC N7:51/1 JSR U:17 EOR
% Rung: 19 %
SOR XIC N7:8/9 XIO N7:8/8 XIC N7:51/1 JSR U:18 EOR
% Rung: 20 %
SOR XIC N7:8/10 XIC N7:51/1 JSR U:19 EOR
% Rung: 21 %
SOR XIC N7:51/1 JSR U:20 EOR
% Rung: 22 %
SOR XIO N7:8/13 BST XIC N7:51/1 NXB XIC N7:53/6 BND XIO N7:61/0 JSR U:21 EOR

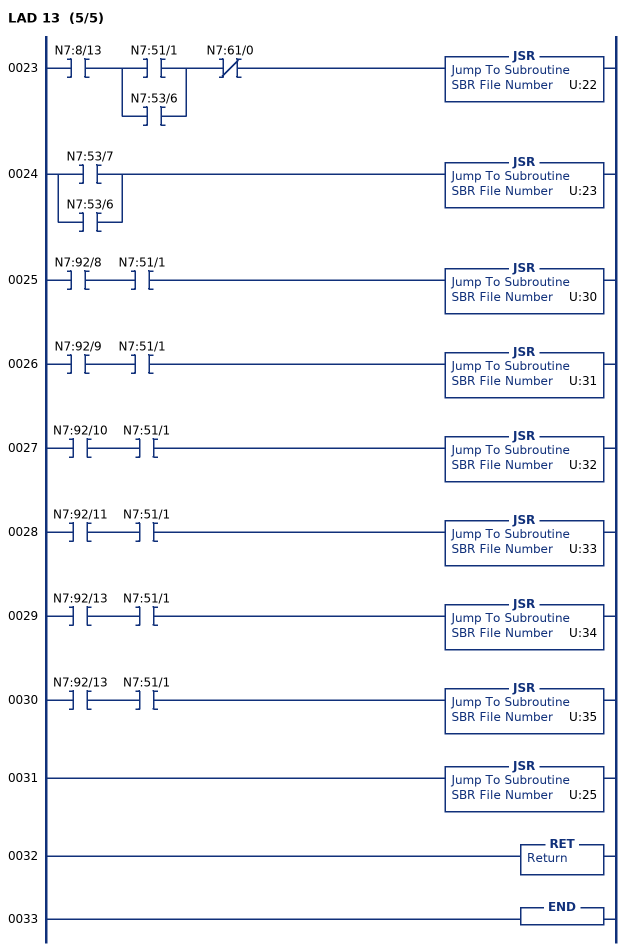
% Rung: 23 %
SOR XIC N7:8/13 BST XIC N7:51/1 NXB XIC N7:53/6 BND XIO N7:61/0 JSR U:22 EOR
% Rung: 24 %
SOR BST XIC N7:53/7 NXB XIC N7:53/6 BND JSR U:23 EOR
% Rung: 25 %
SOR XIC N7:92/8 XIC N7:51/1 JSR U:30 EOR
% Rung: 26 %
SOR XIC N7:92/9 XIC N7:51/1 JSR U:31 EOR
% Rung: 27 %
SOR XIC N7:92/10 XIC N7:51/1 JSR U:32 EOR
% Rung: 28 %
SOR XIC N7:92/11 XIC N7:51/1 JSR U:33 EOR
% Rung: 29 %
SOR XIC N7:92/13 XIC N7:51/1 JSR U:34 EOR
% Rung: 30 %
SOR XIC N7:92/13 XIC N7:51/1 JSR U:35 EOR
% Rung: 31 %
SOR JSR U:25 EOR
% Rung: 32 %
SOR RET EOR
% Rung: 33 %
SOR END EOR

LADDER 14
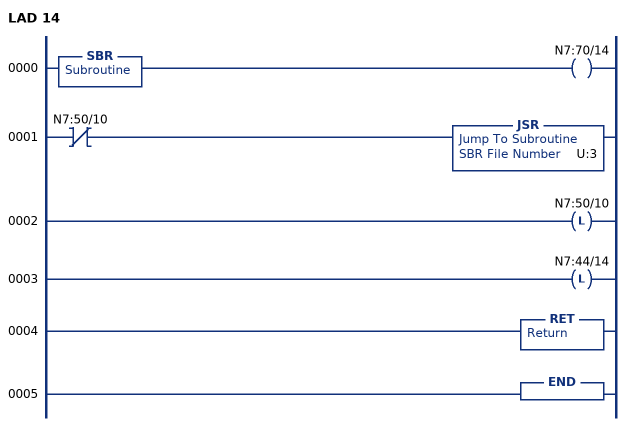
% Rung: 0 %
SOR SBR OTE N7:70/14 EOR
% Rung: 1 %
SOR XIO N7:50/10 JSR U:3 EOR
% Rung: 2 %
SOR OTL N7:50/10 EOR
% Rung: 3 %
SOR OTL N7:44/14 EOR
% Rung: 4 %
SOR RET EOR
% Rung: 5 %
SOR END EOR

LADDER 15
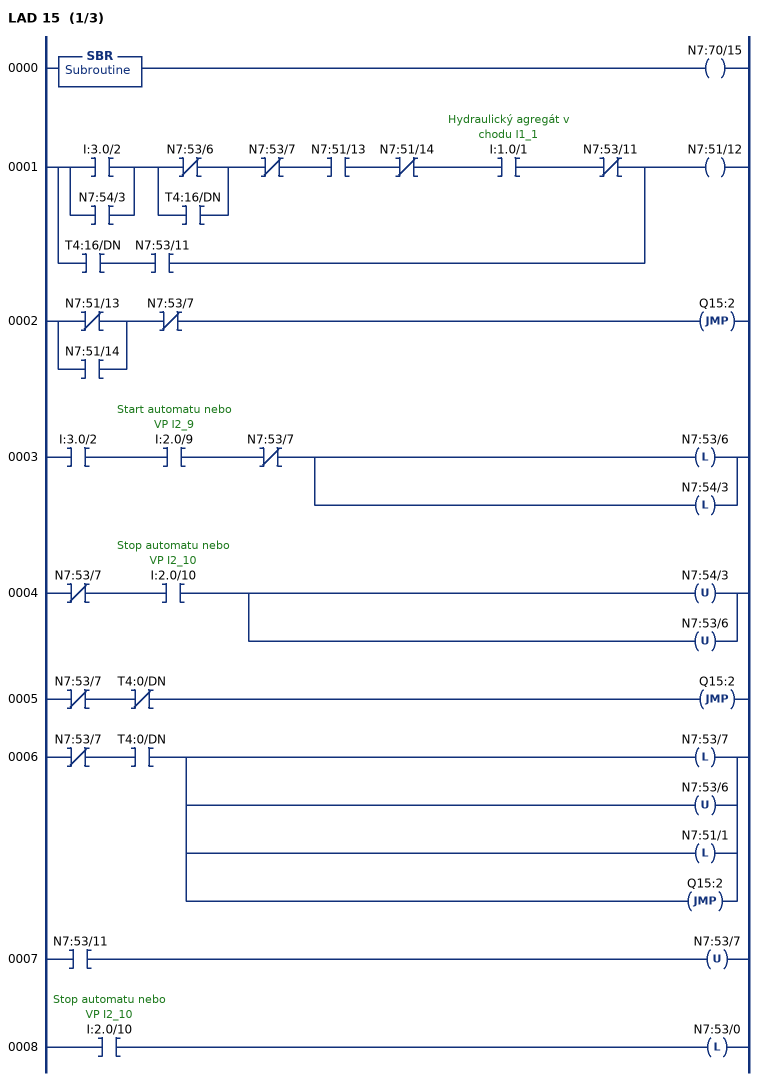
% Rung: 0 %
SOR SBR OTE N7:70/15 EOR
% Rung: 1 %
SOR BST BST XIC I:3.0/2 NXB XIC N7:54/3 BND BST XIO N7:53/6 NXB XIC T4:16/DN BND XIO N7:53/7 XIC N7:51/13 XIO N7:51/14 XIC I:1.0/1 XIO N7:53/11 NXB XIC T4:16/DN XIC N7:53/11 BND OTE N7:51/12 EOR
%   I:1.0/1  I1_1  "Hydraulický agregát v chodu" %
% Rung: 2 %
SOR BST XIO N7:51/13 NXB XIC N7:51/14 BND XIO N7:53/7 JMP Q15:2 EOR
% Rung: 3 %
SOR XIC I:3.0/2 XIC I:2.0/9 XIO N7:53/7 BST OTL N7:53/6 NXB OTL N7:54/3 BND EOR
%   I:2.0/9  I2_9  "Start automatu nebo VP" %
% Rung: 4 %
SOR XIO N7:53/7 XIC I:2.0/10 BST OTU N7:54/3 NXB OTU N7:53/6 BND EOR
%   I:2.0/10  I2_10  "Stop automatu nebo VP" %
% Rung: 5 %
SOR XIO N7:53/7 XIO T4:0/DN JMP Q15:2 EOR
% Rung: 6 %
SOR XIO N7:53/7 XIC T4:0/DN BST OTL N7:53/7 NXB OTU N7:53/6 NXB OTL N7:51/1 NXB JMP Q15:2 BND EOR
% Rung: 7 %
SOR XIC N7:53/11 OTU N7:53/7 EOR
% Rung: 8 %
SOR XIC I:2.0/10 OTL N7:53/0 EOR
%   I:2.0/10  I2_10  "Stop automatu nebo VP" %

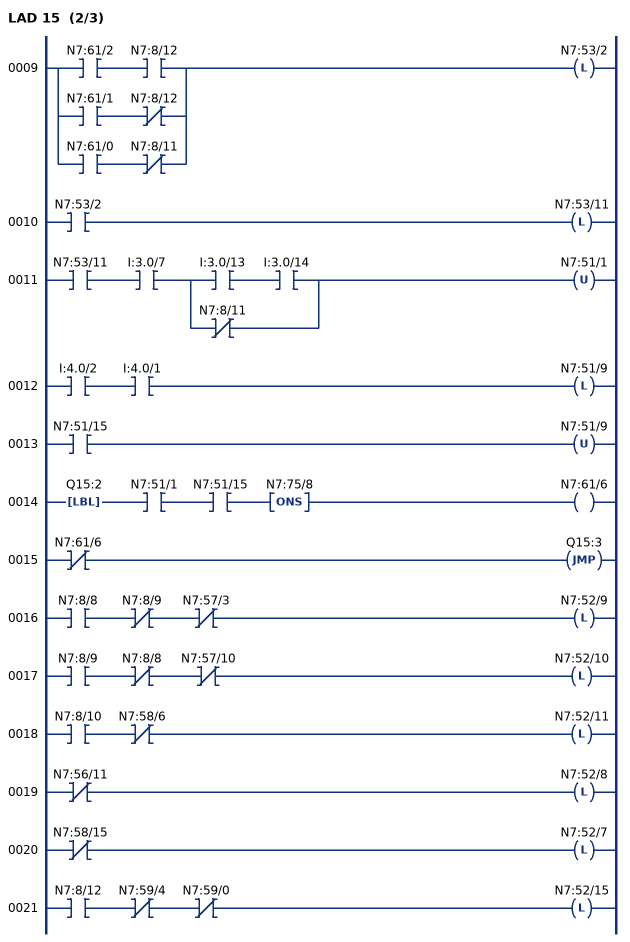
% Rung: 9 %
SOR BST XIC N7:61/2 XIC N7:8/12 NXB XIC N7:61/1 XIO N7:8/12 NXB XIC N7:61/0 XIO N7:8/11 BND OTL N7:53/2 EOR
% Rung: 10 %
SOR XIC N7:53/2 OTL N7:53/11 EOR
% Rung: 11 %
SOR XIC N7:53/11 XIC I:3.0/7 BST XIC I:3.0/13 XIC I:3.0/14 NXB XIO N7:8/11 BND OTU N7:51/1 EOR
% Rung: 12 %
SOR XIC I:4.0/2 XIC I:4.0/1 OTL N7:51/9 EOR
% Rung: 13 %
SOR XIC N7:51/15 OTU N7:51/9 EOR
% Rung: 14 %
SOR LBL Q15:2 XIC N7:51/1 XIC N7:51/15 OSR N7:75/8 OTE N7:61/6 EOR
% Rung: 15 %
SOR XIO N7:61/6 JMP Q15:3 EOR
% Rung: 16 %
SOR XIC N7:8/8 XIO N7:8/9 XIO N7:57/3 OTL N7:52/9 EOR
% Rung: 17 %
SOR XIC N7:8/9 XIO N7:8/8 XIO N7:57/10 OTL N7:52/10 EOR
% Rung: 18 %
SOR XIC N7:8/10 XIO N7:58/6 OTL N7:52/11 EOR
% Rung: 19 %
SOR XIO N7:56/11 OTL N7:52/8 EOR
% Rung: 20 %
SOR XIO N7:58/15 OTL N7:52/7 EOR
% Rung: 21 %
SOR XIC N7:8/12 XIO N7:59/4 XIO N7:59/0 OTL N7:52/15 EOR

